PROGRAM PRG_Compilation
VAR
	fbLoggerElement				: FB_BaseLoggerElement;
	fbLoggerElementDecorator	: FB_BaseLoggerElementDecoratorParent (fbToDecorate := fbLoggerElement);
END_VAR

END_PROGRAM

(* stored: Version 1.1.0.1, ProductVersion 3.1.4024.15
   POU PRG_Compilation: Id {824d9806-ef98-4594-8f89-7dfa640c0d27}, SpecialFunc None *)
